// TIA Portal V21 export
DATA_BLOCK "DB624"   // DB624
{ S7_Optimized_Access := 'FALSE' }
// stored: AutoNumber false
   VAR RETAIN
      PcdTime : Int := 10;
      VesselDrainWeight : Real := 15.0;
      AirPurgingPressureTolerence : Real := 0.1;
      AirPurgingReleaseTime : Int := 30;
      DrainPressureTolerance : Real := 0.2;
      DelayToCheckConductivity : Int := 10;
      ConductivityCheckTime : Int := 5;
      "FinalRinseCycleNo.OfRep" : Int := 3;
      FillRinseSamplingLineDelay : Int := 30;
      FillRinseBlanketingLineDelay : Int := 30;
      FillRinseJTubeLineDelay : Int := 30;
      FillRinseSpargingLineDelay : Int := 30;
      FillRinseSbiLineDelay : Int := 30;
      FillRinseRecirculationlineDelay : Int := 30;
      FillRinseVesselBypassLineDelay : Int := 30;
      FillRinsePumpBypassLineDelay : Int := 30;
      FillRinsePf01InLineDelay : Int := 30;
      FillRinsePf01VentLineDelay : Int := 30;
      FillRinsePf02InLineDelay : Int := 30;
      FillRinsePf02VentLineDelay : Int := 30;
      FillRinsePf02OutLineDelay : Int := 30;
      FillRinsePf01BypassLineDelay : Int := 30;
      FillRinsePf02BypassLineDelay : Int := 30;
      FillRinsePtlLineDelay : Int := 30;
      RecSamplingLineDelay : Int := 30;
      RecBlanketingLineDelay : Int := 30;
      RecJTubeLineDelay : Int := 30;
      RecSpargingLineDelay : Int := 30;
      RecSbiLineDelay : Int := 30;
      DrainVesselDrainLineDelay : Int := 30;
      DrainPumpBypassLineDelay : Int := 30;
      DrainPf01InLineDelay : Int := 30;
      DrainPf01VentLineDelay : Int := 30;
      DrainPf02InLineDelay : Int := 30;
      DrainPf02VentLineDelay : Int := 30;
      DrainPf02OutLineDelay : Int := 30;
      DrainPf01BypassLineDelay : Int := 30;
      DrainPf02BypassLineDelay : Int := 30;
      FinalRinseCycleVesselDrainLineDelay : Int := 30;
      AirPurgeSamplingLineDelay : Int := 30;
      AirPurgeBlankeingLineDelay : Int := 30;
      AirPurgeJTubeLineDelay : Int := 30;
      AirPurgeSpargingLineDelay : Int := 30;
      AirPurgeSbiLineDelay : Int := 30;
      AirPurgeRecirculationlineDelay : Int := 30;
      AirPurgeVesselBypassLineDelay : Int := 30;
      AirPurgeVesselDrainLineDelay : Int := 30;
      AirPurgePumpBypassLineDelay : Int := 30;
      AirPurgePf01InLineDelay : Int := 30;
      AirPurgePf01VentLineDelay : Int := 30;
      AirPurgePf02InLineDelay : Int := 30;
      AirPurgePf02VentLineDelay : Int := 30;
      AirPurgePf02OutLineDelay : Int := 30;
      AirPurgePf01BypassLineDelay : Int := 30;
      AirPurgePf02BypassLineDelay : Int := 30;
      AirPurgePtlLineDelay : Int := 30;
   END_VAR
BEGIN
END_DATA_BLOCK
